# EPICS autosave request: soft_iocs/meas_comp/iocBoot/iocmeas_comp_ctr/auto_settings.req
file "USBCTR_settings.req", P=$(P1), SP=$(P1), MP=$(MP1)
file "USBCTR_settings.req", P=$(P2), SP=$(P2), MP=$(MP2)
file standardScans_settings.req P=$(SP)
file saveData_settings.req P=$(SP)
file "dark.req", P=$(P1)
file "dark.req", P=$(P2)
